// TIA Portal V20 export
VAR_GLOBAL   // PLC tag table "ConvConstantProductionLine"
END_VAR
VAR_GLOBAL CONSTANT   // user constants
   minProductionLine : Int := 1001;
   maxProductionLine : Int := 1192;
   "A1.1.1" : Int := 1001;
   "A1.1.2" : Int := 1002;
   "A1.1.3" : Int := 1003;
   "A1.1.4" : Int := 1004;
   "A1.1.5" : Int := 1005;
   "A1.1.6" : Int := 1006;
   "A1.1.7" : Int := 1007;
   "A1.1.8" : Int := 1008;
   "A1.1.9" : Int := 1009;
   "A1.1.10" : Int := 1010;
   "A1.1.11" : Int := 1011;
   "A1.1.12" : Int := 1012;
   "A1.1.13" : Int := 1013;
   "A1.1.14" : Int := 1014;
   "A1.2.1" : Int := 1015;   // //A1.2.1 (DP1)
   "A1.3.1" : Int := 1016;
   "A1.4.1" : Int := 1017;
   "A1.5.1" : Int := 1018;
   "A1.5.2" : Int := 1019;
   "A1.5.3" : Int := 1020;
   "A1.7.1" : Int := 1021;   // // A1.7.1 (Go Straight DP1)
   "A1.7.2" : Int := 1022;   // //A1.7.2 Straight for Merger1
   "A1.7.3" : Int := 1023;
   "A1.7.4" : Int := 1024;   // //A1.7.4 (DP4)
   "A1.7.5" : Int := 1025;
   "A1.7.6" : Int := 1026;
   "A1.8.1" : Int := 1027;
   "A1.10.1" : Int := 1028;   // // A1.9.1 (Go Straight DP4)
   "A1.10.2" : Int := 1029;   // //A1.9.2 Straight for Merger2
   "A1.10.3" : Int := 1030;   // // A1.9.3 Merger2
   "A1.10.4" : Int := 1031;
   "A1.10.5" : Int := 1032;
   "A1.10.6" : Int := 1033;
   "A1.10.7" : Int := 1034;
   "A1.10.8" : Int := 1035;
   "A1.10.9" : Int := 1036;
   "A1.10.10" : Int := 1037;
   "A1.10.11" : Int := 1038;
   "A1.10.12" : Int := 1039;
   "A1.10.13" : Int := 1040;
   "A1.11.1" : Int := 1041;
   "A1.11.2" : Int := 1042;
   "A1.12.1" : Int := 1043;
   "A1.12.2" : Int := 1044;
   "A1.14.1" : Int := 1045;   // // A1.13.1 (Go straight TR_A1.12.1)
   "A1.14.2" : Int := 1046;
   "A1.14.3" : Int := 1047;
   "A1.14.4" : Int := 1048;
   "A1.14.5" : Int := 1049;
   "A1.14.6" : Int := 1050;
   "A1.14.7" : Int := 1051;
   "A1.14.8" : Int := 1052;
   "A1.14.9" : Int := 1053;
   "A1.14.10" : Int := 1054;
   "A1.14.11" : Int := 1055;
   "A1.14.12" : Int := 1056;
   "A1.14.13" : Int := 1057;
   "A1.14.14" : Int := 1058;
   "A1.14.15" : Int := 1059;
   "A2.2.1" : Int := 1071;   // // A1.17.2 (Go straight TR_A2.1.1)
   "A2.2.2" : Int := 1072;
   "A2.2.3" : Int := 1073;
   "A2.2.4" : Int := 1074;
   "A2.2.5" : Int := 1075;
   "A2.2.6" : Int := 1076;
   "A2.2.7" : Int := 1077;
   "A2.2.8" : Int := 1078;
   "A2.2.9" : Int := 1079;
   "A2.2.10" : Int := 1080;
   "A2.2.11" : Int := 1081;
   "A2.2.12" : Int := 1082;
   "A2.2.13" : Int := 1083;
   "A2.2.14" : Int := 1084;
   "A2.2.15" : Int := 1085;
   "B1.1.1" : Int := 1097;   // // B1.1.1 (Go Right DP1)
   "B1.2.1" : Int := 1098;
   "B1.3.1" : Int := 1099;
   "B1.3.2" : Int := 1100;
   "B1.3.3" : Int := 1101;
   "B1.4.1" : Int := 1102;
   "B1.4.2" : Int := 1103;
   "B1.5.1" : Int := 1104;
   "B1.7.1" : Int := 1105;   // // B1.7.1 (Go straight TR_A1.7.1)
   "B1.7.2" : Int := 1106;
   "B1.7.3" : Int := 1107;
   "B1.8.1" : Int := 1108;
   "B1.8.2" : Int := 1109;
   "B1.8.3" : Int := 1110;
   "B1.9.1" : Int := 1111;   // // B1.9.1 (DP2)
   "B1.9.2" : Int := 1112;
   "B1.11.1" : Int := 1113;   // // B1.11.1 (Go straight TR_B1.11.1)
   "B1.11.2" : Int := 1114;
   "B1.11.3" : Int := 1115;
   "B1.11.4" : Int := 1116;
   "B1.12.1" : Int := 1117;
   "B1.12.2" : Int := 1118;
   "B1.15.1" : Int := 1119;   // // B1.18.1 (Go straight TR_B1.17.1)
   "B1.15.2" : Int := 1120;
   "B1.16.1" : Int := 1121;
   "B1.16.2" : Int := 1122;
   "B1.16.3" : Int := 1123;
   "B1.16.4" : Int := 1124;
   "B1.16.5" : Int := 1125;
   "B1.16.6" : Int := 1126;
   "B1.16.7" : Int := 1127;
   "B1.16.8" : Int := 1128;
   "B1.17.1" : Int := 1129;   // // B1.20.1 (DP3)
   "B1.17.2" : Int := 1130;
   "B1.17.3" : Int := 1131;
   "B1.17.4" : Int := 1132;
   "B1.19.1" : Int := 1133;
   "B1.20.1" : Int := 1134;
   "B1.20.2" : Int := 1135;
   "B1.21.1" : Int := 1136;
   "B1.21.2" : Int := 1137;
   "B1.21.3" : Int := 1138;
   "B1.22.1" : Int := 1139;
   "B1.23.1" : Int := 1140;   // //B1.28.1 Arm for Merger1
   "C1.2.2" : Int := 1141;   // // C1.1.2 (Go Right TR_C1.1.3)
   "C1.2.1" : Int := 1142;
   "C1.4.1" : Int := 1143;   // // C1.1.4 (Go Left TR_C1.1.3)
   "C1.4.2" : Int := 1144;
   "D1.1.1" : Int := 1145;   // // D1.1.1 (Go Right DP4)
   "D1.2.1" : Int := 1146;
   "D1.3.1" : Int := 1147;
   "D1.4.1" : Int := 1148;
   "D1.5.1" : Int := 1149;
   "D1.6.1" : Int := 1150;
   "D1.7.1" : Int := 1151;
   "D1.7.2" : Int := 1152;
   "D1.7.3" : Int := 1153;
   "D1.7.4" : Int := 1154;
   "D1.7.5" : Int := 1155;
   "D1.7.6" : Int := 1156;
   "D1.7.7" : Int := 1157;
   "D1.7.8" : Int := 1158;
   "D1.7.9" : Int := 1159;
   "D1.7.10" : Int := 1160;
   "D1.8.1" : Int := 1161;
   "D1.8.2" : Int := 1162;
   "D1.8.3" : Int := 1163;
   "D1.11.1" : Int := 1164;
   "D1.11.2" : Int := 1165;
   "D1.11.3" : Int := 1166;
   "D1.12.1" : Int := 1167;
   "D1.12.2" : Int := 1168;
   "D1.12.3" : Int := 1169;   // //End
   "E1.1.2" : Int := 1171;
   "E1.1.3" : Int := 1172;
   "E1.1.4" : Int := 1173;
   "E1.2.1" : Int := 1174;
   "E1.3.1" : Int := 1175;
   "E1.4.1" : Int := 1176;
   "E1.5.1" : Int := 1177;
   "E1.6.1" : Int := 1178;   // //E1.6.1 Arm for Merger2
   "A1.9.1" : Int := 1179;   // // Mabs A1.8.1
   "A1.9.2" : Int := 1180;   // // Mabs A1.8.2
   "A1.6.1" : Int := 1181;   // // Mabs A1.6.1
   "A1.6.2" : Int := 1182;   // // Mabs A1.6.2
   "A1.13.1" : Int := 1183;   // // Transfer A1.12.1
   "A2.1.1" : Int := 1184;   // // Transfer A2.1.1
   "B1.6.1" : Int := 1185;   // // Transfer B1.6.1
   "B1.10.1" : Int := 1186;   // // Transfer B1.10.1
   "B1.13.1" : Int := 1187;   // // Transfer B1.16.1
   "B1.14.1" : Int := 1188;   // // Transfer B1.17.1
   "B1.18.1" : Int := 1189;   // // Transfer B1.21.1
   "C1.3.1" : Int := 1190;   // //Transfer C1.1.3
   "D1.9.1" : Int := 1191;   // //Transfer D1.8.1
   "D1.10.1" : Int := 1192;   // //Transfer D1.9.1
   "A1.14.16" : Int := 1060;
   "A1.14.17" : Int := 1061;
   "A1.14.18" : Int := 1062;
   "A1.14.19" : Int := 1063;
   "A1.14.20" : Int := 1064;
   "A1.14.21" : Int := 1065;
   "A1.14.22" : Int := 1066;
   "A1.14.23" : Int := 1067;
   "A1.14.24" : Int := 1068;
   "A2.2.16" : Int := 1086;
   "A2.2.17" : Int := 1087;
   "A2.2.18" : Int := 1088;
   "A2.2.19" : Int := 1089;
   "A2.2.20" : Int := 1090;
   "A2.2.21" : Int := 1091;
   "A2.2.22" : Int := 1092;
   "A2.2.23" : Int := 1093;
   "A2.2.24" : Int := 1094;
   "E1.1.1" : Int := 1170;
   "A1.14.25" : Int := 1069;
   "A1.14.26" : Int := 1070;
   "A2.2.25" : Int := 1095;
   "A2.2.26" : Int := 1096;
END_VAR
